// TIA Portal V17 export
// export: Created 2022-07-20T06:59:39.7415014Z, ExportSetting WithDefaults, DisplayName Totally Integrated Automation Portal, DisplayVersion V17, DisplayName TIA Portal Openness, DisplayVersion V17, DisplayName TIA Portal Version Control Interface, DisplayVersion V17, DisplayName SINAMICS Startdrive Advanced, DisplayVersion V17, DisplayName SINAMICS Startdrive G130, G150, S120, S150, SINAMICS MV, S210, DisplayVersion V17, DisplayName SINAMICS Startdrive G110M, G120, G120C, G120D, G120P, G115D, DisplayVersion V17, DisplayName STEP 7 Professional, DisplayVersion V17, DisplayName STEP 7 Safety, DisplayVersion V17, DisplayName WinCC Advanced, DisplayVersion V17
FUNCTION "FC10017_WordTo2Bytes" : Void   // FC10017, LAD
{ S7_Optimized_Access := 'TRUE' }
VERSION : 0.1
// stored: AutoNumber false, IsIECCheckEnabled false, SetENOAutomatically false, UDAEnableTagReadback false
   VAR_INPUT
      "Word" : Word;
   END_VAR
   VAR_OUTPUT
      HighByte : Byte;
      LowByte : Byte;
   END_VAR
BEGIN

REGION Network 1 (SCL): Conversion Management
   //Low Byte Management
   #LowByte.%X0 := #Word.%X0;
   #LowByte.%X1 := #Word.%X1;
   #LowByte.%X2 := #Word.%X2;
   #LowByte.%X3 := #Word.%X3;
   #LowByte.%X4 := #Word.%X4;
   #LowByte.%X5 := #Word.%X5;
   #LowByte.%X6 := #Word.%X6;
   #LowByte.%X7 := #Word.%X7;

   //High Byte Management
   #HighByte.%X0 := #Word.%X8;
   #HighByte.%X1 := #Word.%X9;
   #HighByte.%X2 := #Word.%X10;
   #HighByte.%X3 := #Word.%X11;
   #HighByte.%X4 := #Word.%X12;
   #HighByte.%X5 := #Word.%X13;
   #HighByte.%X6 := #Word.%X14;
   #HighByte.%X7 := #Word.%X15;
END_REGION
END_FUNCTION
